// TwinCAT 3 PLC project HelloWorld
// ProgramVersion: 3.1.4023.0
// libraries:
//   Tc2_Math, * (Beckhoff Automation GmbH)
//   Tc2_Standard, * (Beckhoff Automation GmbH)
//   Tc2_System, * (Beckhoff Automation GmbH)
//   Tc2_Utilities, * (Beckhoff Automation GmbH)
//   Tc3_Module, * (Beckhoff Automation GmbH)
// project tree:
//   DUTs/ E_EventType.TcDUT, ST_Event.TcDUT
//   / PlcTask.TcTTO
//   POUs/ Clesious_to_faringate.TcPOU, MAIN.TcPOU, Test_function_block.TcPOU, UpdateEventTimestampWithSystemTime.TcPOU
// real-time tasks:
//   TASK PlcTask: cycle T#10ms, priority 20, ADS port 350

CONFIGURATION HelloWorld
    RESOURCE PLC ON TwinCAT3
        TASK PlcTask(INTERVAL := T#10ms, PRIORITY := 20);
        PROGRAM MAIN WITH PlcTask : MAIN;
    END_RESOURCE
END_CONFIGURATION

// ---- DUTs/E_EventType.TcDUT
{attribute 'qualified_only'}
{attribute 'strict'}
TYPE E_EventType :
(
	Alarm := 0,
	Message:=1
);
END_TYPE

// ---- DUTs/ST_Event.TcDUT
TYPE ST_Event :
STRUCT
	eEventType: E_EventType;
	eEventSeverity: TcEventSeverity;
	nEventIdentidy: UDINT;
	sEventText: STRING(255);
	dtTimestamp: DATE_AND_TIME;
END_STRUCT
END_TYPE

// ---- POUs/MAIN.TcPOU
PROGRAM MAIN
VAR
	bRunOnlyOnce:BOOL:=FALSE;
	fOneFloat: REAL;
	sThisIsString: STRING;
	nAnInteger: INT;
	
	nReturnedNumberOfBytesForFloat: UDINT;
	nReturnedNumberOfBytesForString: UDINT;
	nReturnedNumberOfBytesForInteher: UDINT;
	stThisIsOurFirstUnstanceOfAStructure: ST_Event;
	bBoolean:BOOL:=FALSE;
END_VAR

IF NOT  bRunOnlyOnce THEN 
    ADSLOGDINT( msgCtrlMask := ADSLOG_MSGTYPE_ERROR OR ADSLOG_MSGTYPE_LOG, 
                    msgFmtStr := 'Hello, World!', dintArg:= 4711);
					bRunOnlyOnce:=TRUE;
END_IF	  
nReturnedNumberOfBytesForFloat:=SIZEOF(fOneFloat);
nReturnedNumberOfBytesForString:=SIZEOF(sThisIsString);
nReturnedNumberOfBytesForInteher:=SIZEOF(nAnInteger);

IF NOT bBoolean THEN
       UpdateEventTimestampWithSystemTime(stEvent:=stThisIsOurFirstUnstanceOfAStructure);
	   bBoolean:=TRUE;
END_IF;

END_PROGRAM

// ---- POUs/UpdateEventTimestampWithSystemTime.TcPOU
FUNCTION UpdateEventTimestampWithSystemTime 
VAR_INPUT
	stEvent: REFERENCE TO ST_Event;
END_VAR
VAR
	fbGETSYSTEMTIME: GETSYSTEMTIME;
	stFileTime: T_FILETIME;
	
END_VAR

fbGETSYSTEMTIME(timeLoDW =>stFileTime.dwHighDateTime,
	           timeHiDW =>stFileTime.dwLowDateTime);
stEvent.dtTimestamp:= FILETIME_TO_DT(fileTime:=stFileTime);

END_FUNCTION

// ---- POUs/Clesious_to_faringate.TcPOU
FUNCTION Clesious_to_faringate : REAL
VAR_INPUT
END_VAR
VAR
END_VAR

END_FUNCTION

// ---- POUs/Test_function_block.TcPOU
FUNCTION_BLOCK Test_function_block
VAR_INPUT
END_VAR
VAR_OUTPUT
END_VAR
VAR
END_VAR

END_FUNCTION_BLOCK
